// TIA Portal V17 export
// export: Created 2026-04-13T11:12:42.2417663Z, ExportSetting WithDefaults, DisplayName Totally Integrated Automation Portal, DisplayVersion V17 Update 4, DisplayName TIA Portal Openness, DisplayVersion V17 Update 4, DisplayName TIA Portal Version Control Interface, DisplayVersion V17, DisplayName SINAMICS Startdrive Advanced, DisplayVersion V17, DisplayName SINAMICS Startdrive G130, G150, S120, S150, SINAMICS MV, S210, DisplayVersion V17, DisplayName SINAMICS Startdrive G110M, G120, G120C, G120D, G120P, G115D, DisplayVersion V17, DisplayName STEP 7 Professional, DisplayVersion V17 Update 4, DisplayName STEP 7 Safety, DisplayVersion V17, DisplayName WinCC Professional, DisplayVersion V17 Update 4
FUNCTION_BLOCK "上升沿"   // FB59, SCL
{ S7_Optimized_Access := 'TRUE' }
VERSION : 0.1
// stored: AutoNumber true, IsIECCheckEnabled false, IsRetainMemResEnabled false, MemoryReserve 100, SetENOAutomatically false, UDAEnableTagReadback false
   VAR_INPUT
      IN : Bool;
   END_VAR
   VAR_IN_OUT
      Q : Bool;
      State : Bool;
   END_VAR
   VAR
      RT1 { S7_SetPoint := 'True'} : R_TRIG;
   END_VAR
BEGIN
   #RT1(CLK := #IN);
   IF #RT1.Q THEN
       #Q := 1;
   END_IF;
   #State := #RT1.Stat_Bit;
END_FUNCTION_BLOCK
